FUNCTION_BLOCK derived1 EXTENDS base implements itf
VAR_INPUT
END_VAR
VAR_OUTPUT
END_VAR
VAR
END_VAR

METHOD ITF_METH : STRING
VAR_INPUT
END_VAR
ITF_METH := 'derived1 itf method';
END_METHOD

METHOD METH : STRING
VAR_INPUT
END_VAR
METH := 'derived1';
END_METHOD

END_FUNCTION_BLOCK

(* stored: Version 1.1.0.1, ProductVersion 3.1.4022.10
   POU derived1: Id {3a957143-d7e5-4c53-995e-192f1163385e}, SpecialFunc None
   Method ITF_METH: Id {7d04ef0c-c37a-4622-9de2-7e0beaac75fe}
   Method METH: Id {6e1e2dac-51f8-47fe-87c4-47921436fec7} *)
